# EPICS autosave request: support/ebrick/2-2-3/iocBoot/iocebrick/autosave/serialLink.req
$(P)$(R)cntl.VAL
$(P)$(R)cntl.DESC
$(P)$(R)data.VAL
$(P)$(R)data.DESC
$(P)$(R)cntlfmt.VAL
$(P)$(R)datafmt.VAL
